TYPE T_Ctrl_SIf_JCL_Cfg :
STRUCT
END_STRUCT
END_TYPE

(* stored: Version 1.1.0.1, ProductVersion 3.1.0.25
   DUT T_Ctrl_SIf_JCL_Cfg: Id {dc83e891-114f-411d-a9f1-53bb5378281f} *)
